LIN {X 0,Y 61.711,Z 607.122,A -85,B 0,C 180,E1 -30585.478,E2 -30585.478} C_VEL
LIN {X 0,Y 71.724,Z 600.776,A -85,B 0,C 180,E1 -30588.489,E2 -30588.489} C_VEL
LIN {X 0,Y 81.857,Z 592.844,A -85,B 0,C 180,E1 -30590.889,E2 -30590.889} C_VEL
LIN {X 0,Y 90.404,Z 584.751,A -85,B 0,C 180,E1 -30592.397,E2 -30592.397} C_VEL
LIN {X 0,Y 99.006,Z 574.873,A -85,B 0,C 180,E1 -30593.627,E2 -30593.627} C_VEL
LIN {X 0,Y 105.907,Z 565.141,A -85,B 0,C 180,E1 -30594.514,E2 -30594.514} C_VEL
LIN {X 0,Y 111.968,Z 554.581,A -85,B 0,C 180,E1 -30595.174,E2 -30595.174} C_VEL
LIN {X 0,Y 117.486,Z 542.178,A -85,B 0,C 180,E1 -30595.739,E2 -30595.739} C_VEL
LIN {X 0,Y 120.92,Z 531.876,A -85,B 0,C 180,E1 -30596.195,E2 -30596.195} C_VEL
LIN {X 0,Y 121.07,Z 530.606,A -85,B 0,C 180,E1 -30600,E2 -30600} C_VEL
LIN {X 0,Y 120.959,Z 531.95,A -85,B 0,C 180,E1 -30603.523,E2 -30603.523} C_VEL
LIN {X 0,Y 116.625,Z 544.63,A -85,B 0,C 180,E1 -30603.91,E2 -30603.91} C_VEL
LIN {X 0,Y 111.02,Z 556.641,A -85,B 0,C 180,E1 -30604.402,E2 -30604.402} C_VEL
LIN {X 0,Y 104.068,Z 568.173,A -85,B 0,C 180,E1 -30605.043,E2 -30605.043} C_VEL
LIN {X 0,Y 96.265,Z 578.561,A -85,B 0,C 180,E1 -30605.878,E2 -30605.878} C_VEL
LIN {X 0,Y 88.501,Z 587.056,A -85,B 0,C 180,E1 -30606.946,E2 -30606.946} C_VEL
LIN {X 0,Y 78.201,Z 596.263,A -85,B 0,C 180,E1 -30608.658,E2 -30608.658} C_VEL
LIN {X 0,Y 68.017,Z 603.672,A -85,B 0,C 180,E1 -30610.998,E2 -30610.998} C_VEL
LIN {X 0,Y 58.02,Z 609.627,A -85,B 0,C 180,E1 -30614.286,E2 -30614.286} C_VEL
LIN {X 0,Y 48.239,Z 614.33,A -85,B 0,C 180,E1 -30618.732,E2 -30618.732} C_VEL
LIN {X 0,Y 38.876,Z 617.925,A -85,B 0,C 180,E1 -30625.32,E2 -30625.32} C_VEL
LIN {X 0,Y 33.022,Z 619.778,A -85,B 0,C 180,E1 -30631.64,E2 -30631.64} C_VEL
LIN {X 0,Y 23.519,Z 622.171,A -85,B 0,C 180,E1 -30653.294,E2 -30653.294} C_VEL
LIN {X 0,Y 20.748,Z 622.783,A -85,B 0,C 180,E1 -30670.196,E2 -30670.196} C_VEL
LIN {X 0,Y 19.968,Z 622.998,A -85,B 0,C 180,E1 -30689.996,E2 -30689.996} C_VEL
LIN {X 0,Y 20.747,Z 622.762,A -85,B 0,C 180,E1 -30709.797,E2 -30709.797} C_VEL
LIN {X 0,Y 27.808,Z 621.124,A -85,B 0,C 180,E1 -30739.302,E2 -30739.302} C_VEL
LIN {X 0,Y 33.019,Z 619.708,A -85,B 0,C 180,E1 -30748.36,E2 -30748.36} C_VEL
LIN {X 0,Y 41.939,Z 616.756,A -85,B 0,C 180,E1 -30757.169,E2 -30757.169} C_VEL
LIN {X 0,Y 51.476,Z 612.766,A -85,B 0,C 180,E1 -30762.879,E2 -30762.879} C_VEL
LIN {X 0,Y 62.803,Z 606.729,A -85,B 0,C 180,E1 -30767.517,E2 -30767.517} C_VEL
LIN {X 0,Y 73.086,Z 599.938,A -85,B 0,C 180,E1 -30770.275,E2 -30770.275} C_VEL
LIN {X 0,Y 83.334,Z 591.643,A -85,B 0,C 180,E1 -30772.279,E2 -30772.279} C_VEL
LIN {X 0,Y 91.937,Z 583.13,A -85,B 0,C 180,E1 -30773.593,E2 -30773.593} C_VEL
LIN {X 0,Y 100.593,Z 572.617,A -85,B 0,C 180,E1 -30774.608,E2 -30774.608} C_VEL
LIN {X 0,Y 108.407,Z 560.778,A -85,B 0,C 180,E1 -30775.383,E2 -30775.383} C_VEL
LIN {X 0,Y 114.551,Z 548.686,A -85,B 0,C 180,E1 -30775.951,E2 -30775.951} C_VEL
LIN {X 0,Y 119.366,Z 536.118,A -85,B 0,C 180,E1 -30776.338,E2 -30776.338} C_VEL
LIN {X 0,Y 120.686,Z 531.738,A -85,B 0,C 180,E1 -30776.459,E2 -30776.459} C_VEL
LIN {X 0,Y 120.828,Z 530.26,A -85,B 0,C 180,E1 -30780,E2 -30780} C_VEL
LIN {X 0,Y 120.634,Z 531.696,A -85,B 0,C 180,E1 -30783.897,E2 -30783.897} C_VEL
LIN {X 0,Y 116.346,Z 544.263,A -85,B 0,C 180,E1 -30784.428,E2 -30784.428} C_VEL
LIN {X 0,Y 111.11,Z 555.609,A -85,B 0,C 180,E1 -30784.983,E2 -30784.983} C_VEL
LIN {X 0,Y 104.193,Z 567.216,A -85,B 0,C 180,E1 -30785.788,E2 -30785.788} C_VEL
LIN {X 0,Y 96.432,Z 577.649,A -85,B 0,C 180,E1 -30786.792,E2 -30786.792} C_VEL
LIN {X 0,Y 88.707,Z 586.174,A -85,B 0,C 180,E1 -30787.973,E2 -30787.973} C_VEL
LIN {X 0,Y 80.169,Z 594.029,A -85,B 0,C 180,E1 -30789.524,E2 -30789.524} C_VEL
LIN {X 0,Y 70.069,Z 601.693,A -85,B 0,C 180,E1 -30792.06,E2 -30792.06} C_VEL
LIN {X 0,Y 58.426,Z 608.742,A -85,B 0,C 180,E1 -30795.785,E2 -30795.785} C_VEL
LIN {X 0,Y 48.676,Z 613.433,A -85,B 0,C 180,E1 -30800.205,E2 -30800.205} C_VEL
LIN {X 0,Y 39.401,Z 617.015,A -85,B 0,C 180,E1 -30806.896,E2 -30806.896} C_VEL
LIN {X 0,Y 33.855,Z 618.79,A -85,B 0,C 180,E1 -30813.016,E2 -30813.016} C_VEL
LIN {X 0,Y 29.119,Z 620.116,A -85,B 0,C 180,E1 -30818.961,E2 -30818.961} C_VEL
LIN {X 0,Y 24.117,Z 621.104,A -85,B 0,C 180,E1 -30825.537,E2 -30825.537} C_VEL
LIN {X 0,Y 15.108,Z 622.122,A -85,B 0,C 180,E1 -30849.165,E2 -30849.165} C_VEL
LIN {X 0,Y 13.106,Z 622.217,A -85,B 0,C 180,E1 -30872.246,E2 -30872.246} C_VEL
LIN {X 0,Y 13.196,Z 622.15,A -85,B 0,C 180,E1 -30880.921,E2 -30880.921} C_VEL
LIN {X 0,Y 18.725,Z 621.437,A -85,B 0,C 180,E1 -30918.655,E2 -30918.655} C_VEL
LIN {X 0,Y 30.312,Z 619.106,A -85,B 0,C 180,E1 -30938.043,E2 -30938.043} C_VEL
LIN {X 0,Y 39.999,Z 616.232,A -85,B 0,C 180,E1 -30945.111,E2 -30945.111} C_VEL
LIN {X 0,Y 50.073,Z 612.327,A -85,B 0,C 180,E1 -30949.271,E2 -30949.271} C_VEL
LIN {X 0,Y 60.322,Z 607.288,A -85,B 0,C 180,E1 -30952.033,E2 -30952.033} C_VEL
LIN {X 0,Y 71.596,Z 600.267,A -85,B 0,C 180,E1 -30954.366,E2 -30954.366} C_VEL
LIN {X 0,Y 81.035,Z 593.009,A -85,B 0,C 180,E1 -30955.859,E2 -30955.859} C_VEL
LIN {X 0,Y 89.741,Z 584.915,A -85,B 0,C 180,E1 -30956.896,E2 -30956.896} C_VEL
LIN {X 0,Y 98.471,Z 575.036,A -85,B 0,C 180,E1 -30957.728,E2 -30957.728} C_VEL
LIN {X 0,Y 105.466,Z 565.304,A -85,B 0,C 180,E1 -30958.353,E2 -30958.353} C_VEL
LIN {X 0,Y 111.596,Z 554.742,A -85,B 0,C 180,E1 -30958.798,E2 -30958.798} C_VEL
LIN {X 0,Y 117.305,Z 541.995,A -85,B 0,C 180,E1 -30959.202,E2 -30959.202} C_VEL
LIN {X 0,Y 118.638,Z 538.373,A -85,B 0,C 180,E1 -30959.34,E2 -30959.34} C_VEL
LIN {X 0,Y 118.938,Z 537.482,A -85,B 0,C 180,E1 -30959.577,E2 -30959.577} C_VEL
LIN {X 0,Y 118.928,Z 537.521,A -85,B 0,C 180,E1 -30960,E2 -30960} C_VEL
LIN {X 0,Y 118.663,Z 538.323,A -85,B 0,C 180,E1 -30960.282,E2 -30960.282} C_VEL
LIN {X 0,Y 113.841,Z 550.248,A -85,B 0,C 180,E1 -30960.548,E2 -30960.548} C_VEL
LIN {X 0,Y 107.193,Z 562.581,A -85,B 0,C 180,E1 -30960.93,E2 -30960.93} C_VEL
LIN {X 0,Y 99.303,Z 574.069,A -85,B 0,C 180,E1 -30961.417,E2 -30961.417} C_VEL
LIN {X 0,Y 91.421,Z 583.316,A -85,B 0,C 180,E1 -30961.994,E2 -30961.994} C_VEL
LIN {X 0,Y 82.683,Z 591.755,A -85,B 0,C 180,E1 -30962.856,E2 -30962.856} C_VEL
LIN {X 0,Y 72.229,Z 600,A -85,B 0,C 180,E1 -30964.16,E2 -30964.16} C_VEL
LIN {X 0,Y 61.837,Z 606.651,A -85,B 0,C 180,E1 -30966.03,E2 -30966.03} C_VEL
LIN {X 0,Y 49.851,Z 612.733,A -85,B 0,C 180,E1 -30969.29,E2 -30969.29} C_VEL
LIN {X 0,Y 39.724,Z 616.687,A -85,B 0,C 180,E1 -30973.319,E2 -30973.319} C_VEL
LIN {X 0,Y 29.904,Z 619.611,A -85,B 0,C 180,E1 -30979.926,E2 -30979.926} C_VEL
LIN {X 0,Y 18.315,Z 622.004,A -85,B 0,C 180,E1 -30999.865,E2 -30999.865} C_VEL
LIN {X 0,Y 14.253,Z 622.616,A -85,B 0,C 180,E1 -31020.449,E2 -31020.449} C_VEL
LIN {X 0,Y 12.865,Z 622.83,A -85,B 0,C 180,E1 -31049.994,E2 -31049.994} C_VEL
LIN {X 0,Y 14.252,Z 622.594,A -85,B 0,C 180,E1 -31079.541,E2 -31079.541} C_VEL
LIN {X 0,Y 23.783,Z 620.956,A -85,B 0,C 180,E1 -31112.434,E2 -31112.434} C_VEL
LIN {X 0,Y 29.901,Z 619.54,A -85,B 0,C 180,E1 -31120.075,E2 -31120.075} C_VEL
LIN {X 0,Y 39.721,Z 616.587,A -85,B 0,C 180,E1 -31126.684,E2 -31126.684} C_VEL
LIN {X 0,Y 49.847,Z 612.597,A -85,B 0,C 180,E1 -31130.722,E2 -31130.722} C_VEL
LIN {X 0,Y 61.656,Z 606.56,A -85,B 0,C 180,E1 -31133.997,E2 -31133.997} C_VEL
LIN {X 0,Y 72.225,Z 599.768,A -85,B 0,C 180,E1 -31135.85,E2 -31135.85} C_VEL
LIN {X 0,Y 82.679,Z 591.473,A -85,B 0,C 180,E1 -31137.171,E2 -31137.171} C_VEL
LIN {X 0,Y 91.417,Z 582.96,A -85,B 0,C 180,E1 -31138.027,E2 -31138.027} C_VEL
LIN {X 0,Y 100.176,Z 572.447,A -85,B 0,C 180,E1 -31138.656,E2 -31138.656} C_VEL
LIN {X 0,Y 108.067,Z 560.606,A -85,B 0,C 180,E1 -31139.143,E2 -31139.143} C_VEL
LIN {X 0,Y 114.459,Z 548.084,A -85,B 0,C 180,E1 -31139.512,E2 -31139.512} C_VEL
LIN {X 0,Y 118.388,Z 538.124,A -85,B 0,C 180,E1 -31139.703,E2 -31139.703} C_VEL
LIN {X 0,Y 118.698,Z 537.187,A -85,B 0,C 180,E1 -31140,E2 -31140} C_VEL
LIN {X 0,Y 118.716,Z 537.123,A -85,B 0,C 180,E1 -31140.424,E2 -31140.424} C_VEL
LIN {X 0,Y 118.142,Z 538.825,A -85,B 0,C 180,E1 -31140.736,E2 -31140.736} C_VEL
LIN {X 0,Y 113.083,Z 551.066,A -85,B 0,C 180,E1 -31141.126,E2 -31141.126} C_VEL
LIN {X 0,Y 106.343,Z 563.349,A -85,B 0,C 180,E1 -31141.663,E2 -31141.663} C_VEL
LIN {X 0,Y 98.473,Z 574.617,A -85,B 0,C 180,E1 -31142.328,E2 -31142.328} C_VEL
LIN {X 0,Y 89.748,Z 584.567,A -85,B 0,C 180,E1 -31143.218,E2 -31143.218} C_VEL
LIN {X 0,Y 81.041,Z 592.718,A -85,B 0,C 180,E1 -31144.225,E2 -31144.225} C_VEL
LIN {X 0,Y 70.663,Z 600.7,A -85,B 0,C 180,E1 -31145.972,E2 -31145.972} C_VEL
LIN {X 0,Y 60.331,Z 607.104,A -85,B 0,C 180,E1 -31148.049,E2 -31148.049} C_VEL
LIN {X 0,Y 50.084,Z 612.184,A -85,B 0,C 180,E1 -31150.814,E2 -31150.814} C_VEL
LIN {X 0,Y 40.013,Z 616.126,A -85,B 0,C 180,E1 -31154.98,E2 -31154.98} C_VEL
LIN {X 0,Y 30.126,Z 619.073,A -85,B 0,C 180,E1 -31162.175,E2 -31162.175} C_VEL
LIN {X 0,Y 18.723,Z 621.4,A -85,B 0,C 180,E1 -31181.352,E2 -31181.352} C_VEL
LIN {X 0,Y 14.59,Z 622.001,A -85,B 0,C 180,E1 -31201.21,E2 -31201.21} C_VEL
LIN {X 0,Y 13.196,Z 622.15,A -85,B 0,C 180,E1 -31240.921,E2 -31240.921} C_VEL
LIN {X 0,Y 14.636,Z 621.967,A -85,B 0,C 180,E1 -31264.675,E2 -31264.675} C_VEL
LIN {X 0,Y 19.586,Z 621.103,A -85,B 0,C 180,E1 -31293.925,E2 -31293.925} C_VEL
LIN {X 0,Y 25.52,Z 619.907,A -85,B 0,C 180,E1 -31307.301,E2 -31307.301} C_VEL
LIN {X 0,Y 30.768,Z 618.683,A -85,B 0,C 180,E1 -31312.427,E2 -31312.427} C_VEL
LIN {X 0,Y 32.625,Z 618.162,A -85,B 0,C 180,E1 -31313.342,E2 -31313.342} C_VEL
LIN {X 0,Y 42.264,Z 615.197,A -85,B 0,C 180,E1 -31316.169,E2 -31316.169} C_VEL
LIN {X 0,Y 52.747,Z 610.925,A -85,B 0,C 180,E1 -31317.906,E2 -31317.906} C_VEL
LIN {X 0,Y 56.248,Z 609.255,A -85,B 0,C 180,E1 -31318.382,E2 -31318.382} C_VEL
LIN {X 0,Y 56.581,Z 609.11,A -85,B 0,C 180,E1 -31320,E2 -31320} C_VEL
LIN {X 0,Y 45.701,Z 613.998,A -85,B 0,C 180,E1 -31321.581,E2 -31321.581} C_VEL
LIN {X 0,Y 35.222,Z 617.592,A -85,B 0,C 180,E1 -31323.882,E2 -31323.882} C_VEL
LIN {X 0,Y 28.28,Z 619.444,A -85,B 0,C 180,E1 -31326.225,E2 -31326.225} C_VEL
LIN {X 0,Y 14.795,Z 621.837,A -85,B 0,C 180,E1 -31338.171,E2 -31338.171} C_VEL
LIN {X 0,Y 8.797,Z 622.449,A -85,B 0,C 180,E1 -31356.959,E2 -31356.959} C_VEL
LIN {X 0,Y 5.754,Z 622.663,A -85,B 0,C 180,E1 -31409.987,E2 -31409.987} C_VEL
LIN {X 0,Y 8.795,Z 622.427,A -85,B 0,C 180,E1 -31463.031,E2 -31463.031} C_VEL
LIN {X 0,Y 21.433,Z 620.787,A -85,B 0,C 180,E1 -31489.627,E2 -31489.627} C_VEL
LIN {X 0,Y 28.277,Z 619.371,A -85,B 0,C 180,E1 -31493.777,E2 -31493.777} C_VEL
LIN {X 0,Y 38.706,Z 616.418,A -85,B 0,C 180,E1 -31497.001,E2 -31497.001} C_VEL
LIN {X 0,Y 51.829,Z 611.234,A -85,B 0,C 180,E1 -31499.345,E2 -31499.345} C_VEL
LIN {X 0,Y 56.223,Z 609.119,A -85,B 0,C 180,E1 -31500,E2 -31500} C_VEL
LIN {X 0,Y 56.248,Z 609.079,A -85,B 0,C 180,E1 -31501.704,E2 -31501.704} C_VEL
LIN {X 0,Y 45.755,Z 613.769,A -85,B 0,C 180,E1 -31503.271,E2 -31503.271} C_VEL
LIN {X 0,Y 35.32,Z 617.352,A -85,B 0,C 180,E1 -31505.803,E2 -31505.803} C_VEL
LIN {X 0,Y 28.429,Z 619.199,A -85,B 0,C 180,E1 -31508.584,E2 -31508.584} C_VEL
LIN {X 0,Y 15.013,Z 621.567,A -85,B 0,C 180,E1 -31520.581,E2 -31520.581} C_VEL
LIN {X 0,Y 9.042,Z 622.168,A -85,B 0,C 180,E1 -31539.001,E2 -31539.001} C_VEL
LIN {X 0,Y 6.284,Z 622.325,A -85,B 0,C 180,E1 -31610.84,E2 -31610.84} C_VEL
LIN {X 0,Y 15.015,Z 621.604,A -85,B 0,C 180,E1 -31659.425,E2 -31659.425} C_VEL
LIN {X 0,Y 28.428,Z 619.273,A -85,B 0,C 180,E1 -31671.463,E2 -31671.463} C_VEL
LIN {X 0,Y 32.625,Z 618.162,A -85,B 0,C 180,E1 -31673.342,E2 -31673.342} C_VEL
LIN {X 0,Y 32.625,Z 618.162,A -85,B 0,C 180,E1 -31673.342,E2 -31673.342}

QRS_NEXT_CUT()

QRS_NEXT()
QRS_HOME()

END
